DATA_BLOCK "MotorContro_DB_13"
{ S7_Optimized_Access := 'TRUE' }
VERSION : 0.1
NON_RETAIN
// ATTRIBUTES
// AUTO_NUMBER = False
// BLOCK_NUMBER = 3113
// END_ATTRIBUTES
"MotorContro"

BEGIN

END_DATA_BLOCK

